// TIA Portal V20 export
TYPE "LPFE_typeFault"
// stored: Access Published, Namespace PFE
   STRUCT
      Maintenance : Struct
         MF : Struct
            "kDiag.Alarm.AppFault" : Int := 5;   // Logix Programming Faults
            "kDiag.Alarm.LocalIO" : Int := 10;   // Local Chassis Input and Output Card Faults
            "kDiag.Alarm.Power" : Int := 15;   // Power Supply and Circuit Breaker Faults
            "kDiag.Alarm.SafetyComm" : Int := 20;   // Safety Communication Faults
            "kDiag.Alarm.MagnFaults" : Int := 25;   // Relay Faults (abnormal operation)
            "kDiag.Alarm.EStops" : Int := 30;   // Emergency Stop PB and Power Faults
            "kDiag.Alarm.Master" : Int := 35;   // Master On Faults
            "kDiag.Alarm.Comm" : Int := 38;   // Communication Faults
            "kDiag.Alarm.AirAndHyd" : Int := 39;   // Air Pressure and Hydraulic Faults
            "kDiag.Alarm.SwitchFltsBypassable" : Int := 40;   // Switch Faults Bypassable
            "kDiag.Alarm.SwitchFltsNoMotion" : Int := 42;   // Switch Fault No Motion-Not Bypassable
            "kDiag.Alarm.SwitchFltsMotionGrpLimit" : Int := 43;   // Switch Fault Motion Group Limit reached
            "kDiag.Alarm.SwitchFlts" : Int := 44;   // Switch Faults Not Bypassable
            "kDiag.Alarm.VFD" : Int := 48;   // Variable Frequency Drive Faults
            "kDiag.Alarm.PartPres" : Int := 50;   // Part Present Faults
            "kDiag.Alarm.Robots" : Int := 55;   // Robot Faults
            "kDiag.Alarm.Welding" : Int := 60;   // Welding Faults
            "kDiag.Alarm.ProcessEquip" : Int := 65;   // Misc. Process Equipment Faults
            "kDiag.Alarm.Gates" : Int := 75;   // Perimeter Gate Faults
            "kDiag.Alarm.MagnSts" : Int := 80;   // Relay Status
            "kDiag.Alarm.Mode" : Int := 85;   // Automatic Mode Faults
            "kDiag.Alarm.Cycle" : Int := 90;   // Automatic Cycle Faults
            "kDiag.Alarm.Status" : Int := 93;   // Lowest Level Faults
            "kDiag.Alarm.MaintFltAndon" : Int := 97;
         END_STRUCT;
      END_STRUCT;
      Production : Struct
         PF : Struct
            "kDiag.Alarm.ProdFltAndonStop" : Int := 104;   // Production Fault Andon Line Stop
            "kDiag.Alarm.ProdFltOperLoad" : Int := 105;   // Production Fault Operator Load Device
            "kDiag.Alarm.ProdFltAndonEOT" : Int := 106;
            "kDiag.Alarm.ProdFltAndonEStop" : Int := 107;
            "kDiag.Alarm.ProdFltGeneral" : Int := 120;   // Production Fault General
         END_STRUCT;
      END_STRUCT;
      Tooling : Struct
         LF : Struct
            "kDiag.Alarm.ToolFltDimExceeded" : Int := 124;   // Tooling Fault Dimension Exceeded
            "kDiag.Alarm.ToolFltGeneral" : Int := 140;   // Tooling Fault General
         END_STRUCT;
      END_STRUCT;
      Quality : Struct
         QF : Struct
            "kDiag.Alarm.QualFltAndon" : Int := 149;
            "kDiag.Alarm.QualFltGeneral" : Int := 150;   // Quality Fault General
         END_STRUCT;
      END_STRUCT;
      Throughput : Struct
         TFIB : Struct
            "kDiag.Alarm.TputFltBlocked" : Int := 151;   // Thruput Fault Blocked
         END_STRUCT;
         TFS : Struct
            "kDiag.Alarm.TputFltBlockedAndon" : Int := 152;   // Thruput Fault Starved
         END_STRUCT;
         TF : Struct
            "kDiag.Alarm.TputFltBlockedAndon" : Int := 153;
            "kDiag.Alarm.TputFltStarvedAndon" : Int := 154;
            "kDiag.Alarm.TputFltGeneral" : Int := 160;   // Thruput Fault General
         END_STRUCT;
      END_STRUCT;
      System : Struct
         SF : Struct
            "kDiag.Alarm.SysFltGeneral" : Int := 170;   // System Fault General
         END_STRUCT;
      END_STRUCT;
      Material : Struct
         AF : Struct
            "kDiag.Alarm.MatlFltOutOfParts" : Int := 171;   // Material Fault Out of Parts
            "kDiag.Alarm.MatlFltGeneral" : Int := 180;   // Material Fault General
         END_STRUCT;
      END_STRUCT;
   END_STRUCT;
END_TYPE
